(* PLC project Cell Example , CTH FIX1 1.0, author CTH SS2 *)
(* stored: companyURL www.chalmers.se, creationDateTime 2008-03-19T20:31:26, version 1.0, modificationDateTime 2008-04-16T16:39:13, organization SS2, language en-US *)

TYPE BinaryPositions : ();
END_TYPE

FUNCTION_BLOCK RAC
  VAR_INPUT
    IN1 : BOOL := FALSE;
  END_VAR
  VAR_OUTPUT
    OUT : BOOL := FALSE;
  END_VAR
  VAR
    internal : INT := 0;
  END_VAR
  VAR_INPUT
    data : STRING := 'Undefined';
    IN2 : BOOL;
  END_VAR
  VAR
    IN3 : BOOL;
    IN4 : BOOL;
  END_VAR

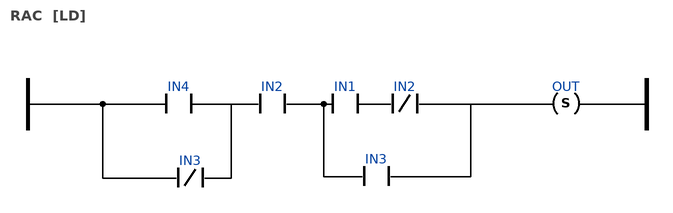
(* LD diagram, written out as Structured Text *)
IF (NOT IN3 OR IN4) AND IN2 AND (IN1 AND NOT IN2 OR IN3) THEN OUT := TRUE; END_IF;
END_FUNCTION_BLOCK

CONFIGURATION ExampleCell
END_CONFIGURATION
